// TIA Portal V20 export
TYPE "typeSequenceControlNodeJobInterface_jrOutPnPRight"
// stored: Namespace Unit1.Em2
   STRUCT
      PICKJob2 : "LER_typeJobInterface";
      PLACEJob3 : "LER_typeJobInterface";
   END_STRUCT;
END_TYPE
